PROGRAM Carriage_Manager_1
VAR
	ResetError: BOOL;
	manager: FB_AchsManager;
	
	Setting: TAxSettingsModule:= (  //the 4 setting itself are general constants that are set at the begining. 
		MaxPos := 100000,
		MinPos := 0,
		Velocity := 250,
		Accel := 250, 
		Deccel := 250	);
	
	Offset: LREAL; //general offset of the encoder value
		
	//half the settings have been filled out already. the FB is used to fill the remaining empty variables. fill out the rest of the starting values up here
	VeloOverride: INT := 100; // usually used to slow the motor
	AccOverride: INT := 100; //acceeration or the over ride
	DccOverride: INT := 100; // deceleration of the override
	JerkOverride: INT := 100; //jerk
	ActivateJogFast: BOOL; //trigger for fast movement
	VeloManJog: REAL := 75; //speed of the regular jog movement
	VeloManJogFAST: REAL := 50; // speed of the fast movement
	AccManJOG: REAL := 50; //general ACC
	DccManJog: REAL := 100; // general DCC
	MaxTorque: WORD := 150; //150% of max torque
	
	
//	Forwards  : BOOL;
	ManConsent: BOOL;
//	Backwards  : BOOL;
	Target: INT;
	RefTrigger: BOOL;
	
	ExtraSensorInput: TAxSensorModule; // compressed FUN for exteriour sensor inputs. temp, edge, jog stops
	SpecialOperations: TAxSpecialOperationModule; //compressed FUN for the special operation commands. 
	AxisCoupleIN: TAxCoupleModule; //connects to the AX_Couple_out of the manager from the next axis. NOT MASTER/SLAVE
	DriveIsReal: BOOL; //a check to make sure the drive is real.
	ErrorWordArray: WORD; //build a array of words that act as a cluster of error watching variables. each step in array will be one axis. differant values of the word for each axis mean a differant error. 
	
	ASP: TASPState; //safety interlock system. connects to the safety program OR build a blank ASP that fills all the values but doesnt connect anywhere. 
	
	TargetPositionActivate: BOOL; //starts the drive positing to the Sollpos
	JogStop: LREAL := 1E100 ; // a stopping point using the jog system to signify it is in the right spot. Need to have the LimitPosJOG adjusted after to compensate for the next space.

	
	(*
	//programed commands for movement and controls. NOT part of the PMA build, this is exteriour controls. 
	
	ManVsAutoSW: BOOL;
	ResetButton: BOOL;
	PHYSICALManVsAutoSW: BOOL;
	
	TON_OKdelay: TON;
	*)
	MotorOK: BOOL; // link this into the EL6910 output STO status. then when STO is good this will be good too. 
	
	StartButton: BOOL;
	
	DriveCMD_1: DriveCMDShortCUT; //extra system for the FB to make it easy to read.
	ASPshortCut_1: ASPshortCUT;  // same as above
	
	ManIN: BOOL;
	AutoIN: BOOL;
	ResetBTN: BOOL;
	SwitchMAN: BOOL;
	SwitchAuto: BOOL;
	AutoRUN: BOOL;
	SafeTEST: BOOL;
END_VAR

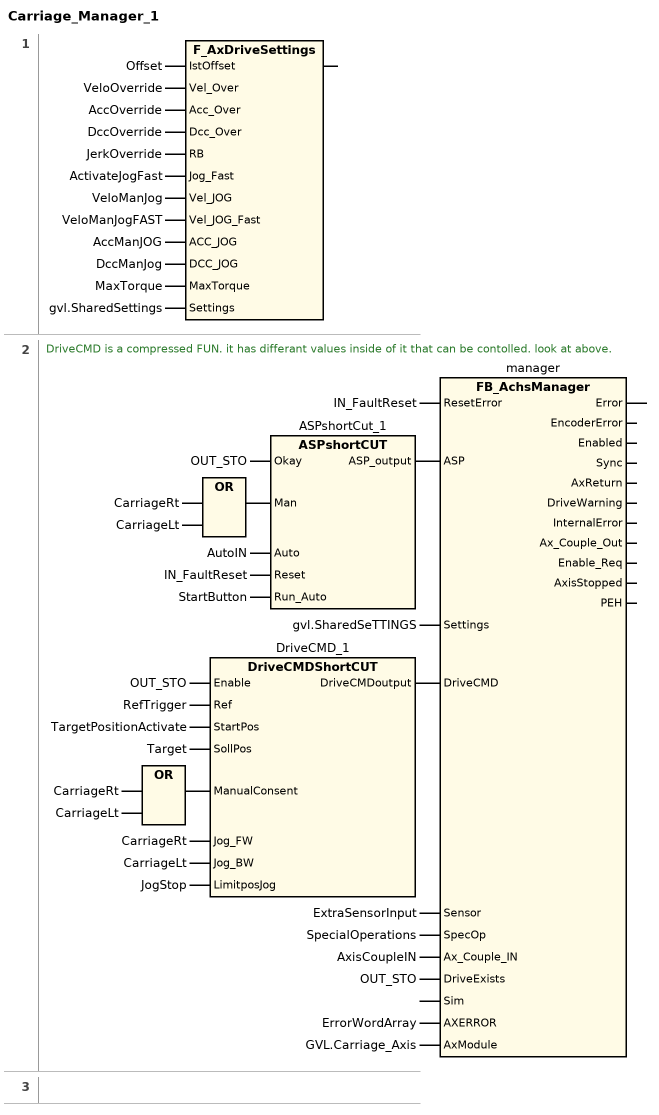
// NETWORK 1
F_AxDriveSettings(IstOffset := Offset, Vel_Over := VeloOverride, Acc_Over := AccOverride, Dcc_Over := DccOverride, RB := JerkOverride, Jog_Fast := ActivateJogFast, Vel_JOG := VeloManJog, Vel_JOG_Fast := VeloManJogFAST, ACC_JOG := AccManJOG, DCC_JOG := DccManJog, MaxTorque := MaxTorque, Settings := gvl.SharedSettings);

// NETWORK 2
// DriveCMD is a compressed FUN. it has differant values inside of it that can be contolled. look at above.
ASPshortCut_1(
    Okay := OUT_STO,
    Man := CarriageRt OR CarriageLt,
    Auto := AutoIN,
    Reset := IN_FaultReset,
    Run_Auto := StartButton); // ASPshortCUT
DriveCMD_1(
    Enable := OUT_STO,
    Ref := RefTrigger,
    StartPos := TargetPositionActivate,
    SollPos := Target,
    ManualConsent := CarriageRt OR CarriageLt,
    Jog_FW := CarriageRt,
    Jog_BW := CarriageLt,
    LimitposJog := JogStop); // DriveCMDShortCUT
manager(
    ResetError := IN_FaultReset,
    ASP := ASPshortCut_1.ASP_output,
    Settings := gvl.SharedSeTTINGS,
    DriveCMD := DriveCMD_1.DriveCMDoutput,
    Sensor := ExtraSensorInput,
    SpecOp := SpecialOperations,
    Ax_Couple_IN := AxisCoupleIN,
    DriveExists := OUT_STO,
    AXERROR := ErrorWordArray,
    AxModule := GVL.Carriage_Axis); // FB_AchsManager

// NETWORK 3

END_PROGRAM

(* stored: Version 1.1.0.1, ProductVersion 3.1.4024.15
   POU Carriage_Manager_1: Id {ce382cb4-b178-4301-a3f0-4db87b1e4dc0}, SpecialFunc None *)
